// TIA Portal project "11_Sorting_Station" (V19)

(* hardware
DEVICE "S7-1500/ET200MP station_1"  S7-1500 station
   slot 0: "Rail_0"  Rack  6ES7 590-1***0-0AA0
   slot 1: "PLC_1"  CPU 1513-1 PN  6ES7 513-1AL02-0AB0  V2.9
      slot 3: "CPU display_1"  6ES7591-1AA00-0AA0
      slot 32768: "PROFINET interface_1"  X1
         slot 32769: "Port_1"  X1 P1
         slot 32770: "Port_2"  X1 P2
      slot 34817: "Virtual CP interface port_1"  Virtual CP interface port  Virtual CP interface port
*)

// ===== PLC "PLC_1"  CPU 1513-1 PN =====

VAR_GLOBAL   // PLC tag table "Default tag table"
   "nw2" AT %M0.0 : Bool;
   "nw3 2nd memory (Pause)" AT %M0.2 : Bool;
   "nw3 1st memory (Unpause)" AT %M0.1 : Bool;
   "nw4" AT %M0.5 : Bool;
   "nw4 Vision sensor O/P" AT %M0.6 : Bool;
   "nw5" AT %M0.3 : Bool;
   "nw5 VS O/P N" AT %M0.7 : Bool;
   "nw6" AT %M0.4 : Bool;
   "nw7" AT %M1.0 : Bool;
   "nw10" AT %M1.3 : Bool;
   "nw10 s1t N" AT %M1.4 : Bool;
   "nw11" AT %M1.5 : Bool;
   "nw11 s2t N" AT %M1.6 : Bool;
   "nw12" AT %M1.7 : Bool;
   "nw12 s2t N" AT %M2.0 : Bool;
   "nw8" AT %M1.1 : Bool;
   "nw9" AT %M1.2 : Bool;
END_VAR

VAR_GLOBAL   // PLC tag table "Tag table from XML_1"
   "Start" AT %I0.0 : Bool;
   "Pause & Unpause" AT %I0.1 : Bool;
   "Reset" AT %I0.2 : Bool;
   "At exit" AT %I0.3 : Bool;
   "Start light" AT %Q0.0 : Bool;
   "Pause & U Light" AT %Q0.1 : Bool;
   "Reset light" AT %Q0.2 : Bool;
   "Entry conveyor" AT %Q0.3 : Bool;
   "Exit conveyor" AT %Q0.4 : Bool;
   "Sorter 1 belt" AT %Q0.5 : Bool;
   "Sorter 1 turn" AT %Q0.6 : Bool;
   "Sorter 2 belt" AT %Q0.7 : Bool;
   "Sorter 2 turn" AT %Q1.0 : Bool;
   "Sorter 3 belt" AT %Q1.1 : Bool;
   "Sorter 3 turn" AT %Q1.2 : Bool;
   "Vision sensor" AT %ID30 : DInt;
   "Raw Materials Count" AT %QD30 : DInt;
   "Product Base Count" AT %QD34 : DInt;
   "Product Lid Count" AT %QD38 : DInt;
END_VAR

// folder: System blocks/Program resources

DATA_BLOCK "IEC_Counter_0_DB"   // DB1
{ S7_Optimized_Access := 'TRUE' }
AUTHOR : Simatic
FAMILY : IEC
NAME : CNTR
VERSION : 1.0
// stored: InstanceOfName IEC_COUNTER
"IEC_COUNTER"
BEGIN
END_DATA_BLOCK

DATA_BLOCK "IEC_Counter_0_DB_1"   // DB2
{ S7_Optimized_Access := 'TRUE' }
AUTHOR : Simatic
FAMILY : IEC
NAME : CNTR
VERSION : 1.0
// stored: InstanceOfName IEC_COUNTER
"IEC_COUNTER"
BEGIN
END_DATA_BLOCK

DATA_BLOCK "IEC_Counter_0_DB_2"   // DB3
{ S7_Optimized_Access := 'TRUE' }
AUTHOR : Simatic
FAMILY : IEC
NAME : CNTR
VERSION : 1.0
// stored: InstanceOfName IEC_COUNTER
"IEC_COUNTER"
BEGIN
END_DATA_BLOCK

// folder: (top level)

ORGANIZATION_BLOCK "Main"   // OB1, LAD, ProgramCycle
TITLE = "Main Program Sweep (Cycle)"
{ S7_Optimized_Access := 'TRUE' }
VERSION : 0.1
   VAR_INPUT
      Initial_Call : Bool;   // Initial call of this OB
      Remanence : Bool;   // =True, if remanent data are available
   END_VAR
   VAR_TEMP   // added for the SCL form of the ladder/FBD networks
      _w1 : Bool;
   END_VAR
BEGIN

REGION Network 2: Start/Reset system
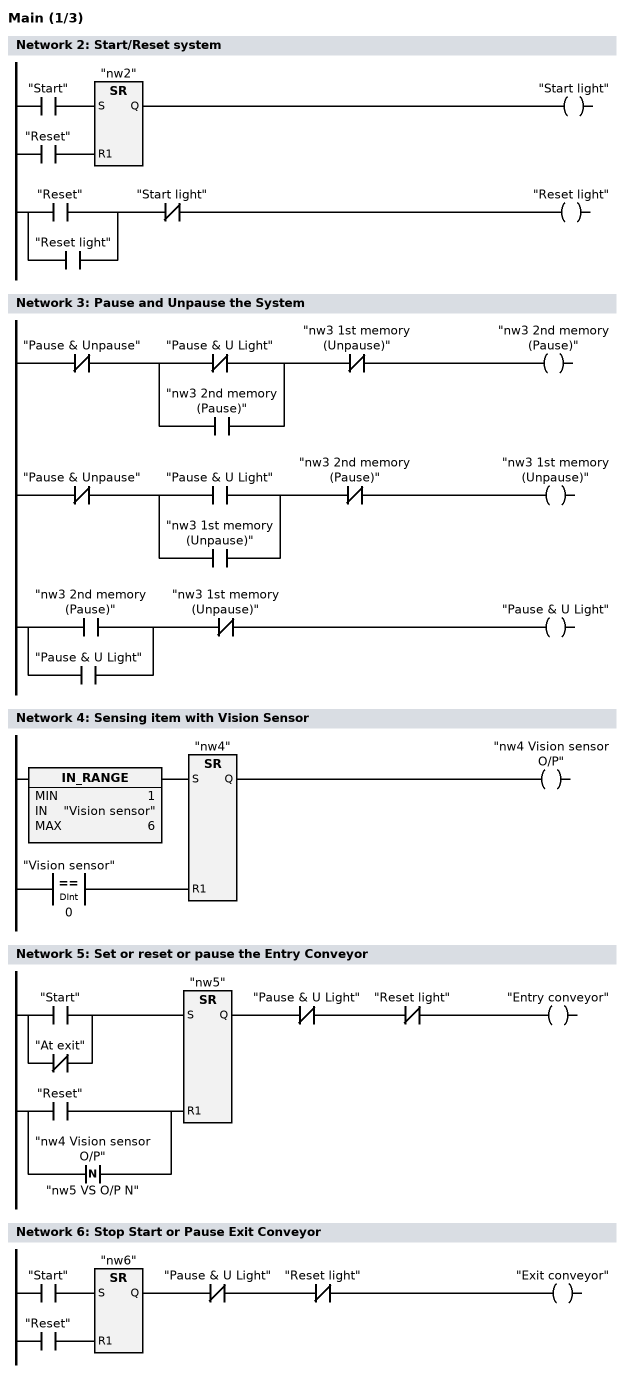
   RUNG wire#powerrail
      Contact( "Start" )
      S_SR(operand := "nw2", r1 := wire#w1)
      Coil( "Start light" )
   END_RUNG
   RUNG wire#powerrail
      Contact( "Reset" )
   END_RUNG wire#w1
   RUNG wire#powerrail
      Contact( "Reset" )
      wire#w2
      I_Contact( "Start light" )
      Coil( "Reset light" )
   END_RUNG
   RUNG wire#powerrail
      Contact( "Reset light" )
   END_RUNG wire#w2
   // the same network as SCL:
   IF "Start" THEN
       "nw2" := TRUE;   // SR flip-flop
   END_IF;
   IF "Reset" THEN "nw2" := FALSE; END_IF;
   "Start light" := "nw2";
   "Reset light" := ("Reset" OR "Reset light") AND NOT "Start light";
END_REGION

REGION Network 3: Pause and Unpause the System
   RUNG wire#powerrail
      I_Contact( "Pause & Unpause" )
      wire#w1
      I_Contact( "Pause & U Light" )
      wire#w2
      I_Contact( "nw3 1st memory (Unpause)" )
      Coil( "nw3 2nd memory (Pause)" )
   END_RUNG
   RUNG wire#w1
      Contact( "nw3 2nd memory (Pause)" )
   END_RUNG wire#w2
   RUNG wire#powerrail
      I_Contact( "Pause & Unpause" )
      wire#w3
      Contact( "Pause & U Light" )
      wire#w4
      I_Contact( "nw3 2nd memory (Pause)" )
      Coil( "nw3 1st memory (Unpause)" )
   END_RUNG
   RUNG wire#w3
      Contact( "nw3 1st memory (Unpause)" )
   END_RUNG wire#w4
   RUNG wire#powerrail
      Contact( "nw3 2nd memory (Pause)" )
      wire#w5
      I_Contact( "nw3 1st memory (Unpause)" )
      Coil( "Pause & U Light" )
   END_RUNG
   RUNG wire#powerrail
      Contact( "Pause & U Light" )
   END_RUNG wire#w5
   // the same network as SCL:
   "nw3 2nd memory (Pause)" := NOT "Pause & Unpause" AND (NOT "Pause & U Light" OR "nw3 2nd memory (Pause)") AND NOT "nw3 1st memory (Unpause)";
   "nw3 1st memory (Unpause)" := NOT "Pause & Unpause" AND ("Pause & U Light" OR "nw3 1st memory (Unpause)") AND NOT "nw3 2nd memory (Pause)";
   "Pause & U Light" := ("nw3 2nd memory (Pause)" OR "Pause & U Light") AND NOT "nw3 1st memory (Unpause)";
END_REGION

REGION Network 4: Sensing item with Vision Sensor
   RUNG wire#powerrail
      { S7_Templates := "SrcType := DInt" } InRange(min := 1, in := "Vision sensor", max := 6)
      S_SR(operand := "nw4", r1 := wire#w1)
      Coil( "nw4 Vision sensor O/P" )
   END_RUNG
   RUNG wire#powerrail
      { S7_Templates := "SrcType := DInt" } EQ_Contact(in1 := "Vision sensor", in2 := 0)
   END_RUNG wire#w1
   // the same network as SCL:
   IF (1 <= "Vision sensor") AND ("Vision sensor" <= 6) THEN
       "nw4" := TRUE;   // SR flip-flop
   END_IF;
   IF "Vision sensor" = 0 THEN "nw4" := FALSE; END_IF;
   "nw4 Vision sensor O/P" := "nw4";
END_REGION

REGION Network 5: Set or reset or pause the Entry Conveyor
   RUNG wire#powerrail
      Contact( "Start" )
      wire#w1
      S_SR(operand := "nw5", r1 := wire#w2)
      I_Contact( "Pause & U Light" )
      I_Contact( "Reset light" )
      Coil( "Entry conveyor" )
   END_RUNG
   RUNG wire#powerrail
      I_Contact( "At exit" )
   END_RUNG wire#w1
   RUNG wire#powerrail
      Contact( "Reset" )
   END_RUNG wire#w2
   RUNG wire#powerrail
      N_Contact(operand := "nw4 Vision sensor O/P", bit := "nw5 VS O/P N")
   END_RUNG wire#w2
   // the same network as SCL:
   #_w1 := NOT "nw4 Vision sensor O/P" AND "nw5 VS O/P N";   // falling edge of "nw4 Vision sensor O/P"
   "nw5 VS O/P N" := "nw4 Vision sensor O/P";
   IF "Start" OR NOT "At exit" THEN
       "nw5" := TRUE;   // SR flip-flop
   END_IF;
   IF "Reset" OR #_w1 THEN "nw5" := FALSE; END_IF;
   "Entry conveyor" := "nw5" AND NOT "Pause & U Light" AND NOT "Reset light";
END_REGION

REGION Network 6: Stop Start or Pause Exit Conveyor
   RUNG wire#powerrail
      Contact( "Start" )
      S_SR(operand := "nw6", r1 := wire#w1)
      I_Contact( "Pause & U Light" )
      I_Contact( "Reset light" )
      Coil( "Exit conveyor" )
   END_RUNG
   RUNG wire#powerrail
      Contact( "Reset" )
   END_RUNG wire#w1
   // the same network as SCL:
   IF "Start" THEN
       "nw6" := TRUE;   // SR flip-flop
   END_IF;
   IF "Reset" THEN "nw6" := FALSE; END_IF;
   "Exit conveyor" := "nw6" AND NOT "Pause & U Light" AND NOT "Reset light";
END_REGION

REGION Network 7: Set/Reset/Pause for Sorter 1, which is RAW_MATERIALS
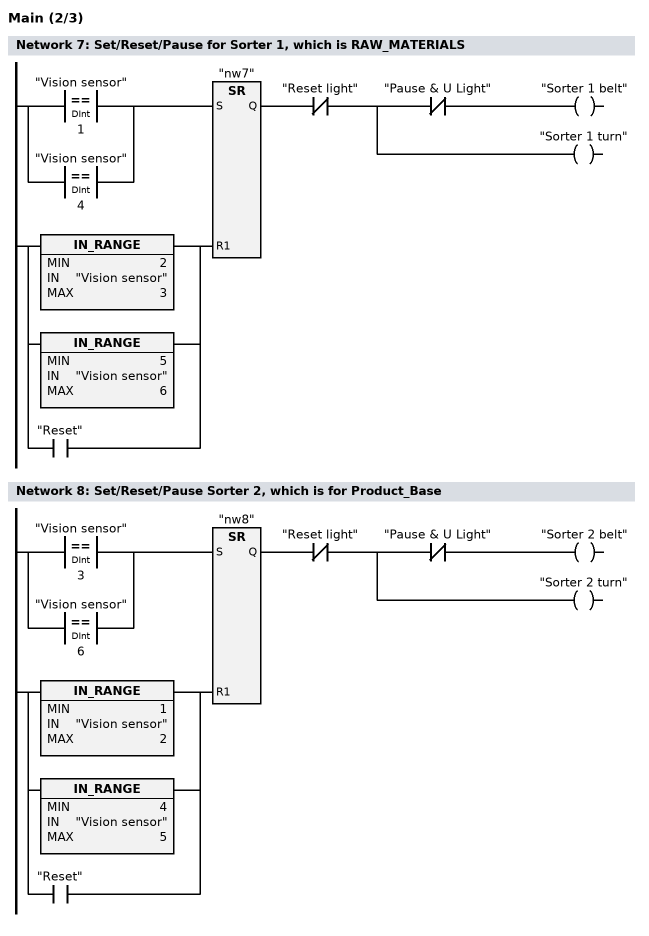
   RUNG wire#powerrail
      { S7_Templates := "SrcType := DInt" } EQ_Contact(in1 := "Vision sensor", in2 := 1)
      wire#w1
      S_SR(operand := "nw7", r1 := wire#w2)
      I_Contact( "Reset light" )
      wire#w3
      I_Contact( "Pause & U Light" )
      Coil( "Sorter 1 belt" )
   END_RUNG
   RUNG wire#powerrail
      { S7_Templates := "SrcType := DInt" } EQ_Contact(in1 := "Vision sensor", in2 := 4)
   END_RUNG wire#w1
   RUNG wire#powerrail
      { S7_Templates := "SrcType := DInt" } InRange(min := 2, in := "Vision sensor", max := 3)
   END_RUNG wire#w2
   RUNG wire#powerrail
      { S7_Templates := "SrcType := DInt" } InRange(min := 5, in := "Vision sensor", max := 6)
   END_RUNG wire#w2
   RUNG wire#powerrail
      Contact( "Reset" )
   END_RUNG wire#w2
   RUNG wire#w3
      Coil( "Sorter 1 turn" )
   END_RUNG
   // the same network as SCL:
   IF ("Vision sensor" = 1) OR ("Vision sensor" = 4) THEN
       "nw7" := TRUE;   // SR flip-flop
   END_IF;
   IF ((2 <= "Vision sensor") AND ("Vision sensor" <= 3)) OR ((5 <= "Vision sensor") AND ("Vision sensor" <= 6)) OR "Reset" THEN
       "nw7" := FALSE;
   END_IF;
   #_w1 := "nw7" AND NOT "Reset light";
   "Sorter 1 belt" := #_w1 AND NOT "Pause & U Light";
   "Sorter 1 turn" := #_w1;
END_REGION

REGION Network 8: Set/Reset/Pause Sorter 2, which is for Product_Base
   RUNG wire#powerrail
      { S7_Templates := "SrcType := DInt" } EQ_Contact(in1 := "Vision sensor", in2 := 3)
      wire#w1
      S_SR(operand := "nw8", r1 := wire#w2)
      I_Contact( "Reset light" )
      wire#w3
      I_Contact( "Pause & U Light" )
      Coil( "Sorter 2 belt" )
   END_RUNG
   RUNG wire#powerrail
      { S7_Templates := "SrcType := DInt" } EQ_Contact(in1 := "Vision sensor", in2 := 6)
   END_RUNG wire#w1
   RUNG wire#powerrail
      { S7_Templates := "SrcType := DInt" } InRange(min := 1, in := "Vision sensor", max := 2)
   END_RUNG wire#w2
   RUNG wire#powerrail
      { S7_Templates := "SrcType := DInt" } InRange(min := 4, in := "Vision sensor", max := 5)
   END_RUNG wire#w2
   RUNG wire#powerrail
      Contact( "Reset" )
   END_RUNG wire#w2
   RUNG wire#w3
      Coil( "Sorter 2 turn" )
   END_RUNG
   // the same network as SCL:
   IF ("Vision sensor" = 3) OR ("Vision sensor" = 6) THEN
       "nw8" := TRUE;   // SR flip-flop
   END_IF;
   IF ((1 <= "Vision sensor") AND ("Vision sensor" <= 2)) OR ((4 <= "Vision sensor") AND ("Vision sensor" <= 5)) OR "Reset" THEN
       "nw8" := FALSE;
   END_IF;
   #_w1 := "nw8" AND NOT "Reset light";
   "Sorter 2 belt" := #_w1 AND NOT "Pause & U Light";
   "Sorter 2 turn" := #_w1;
END_REGION

REGION Network 9: Set/Reset/Pause Sorter 3, which is for Product_Lid
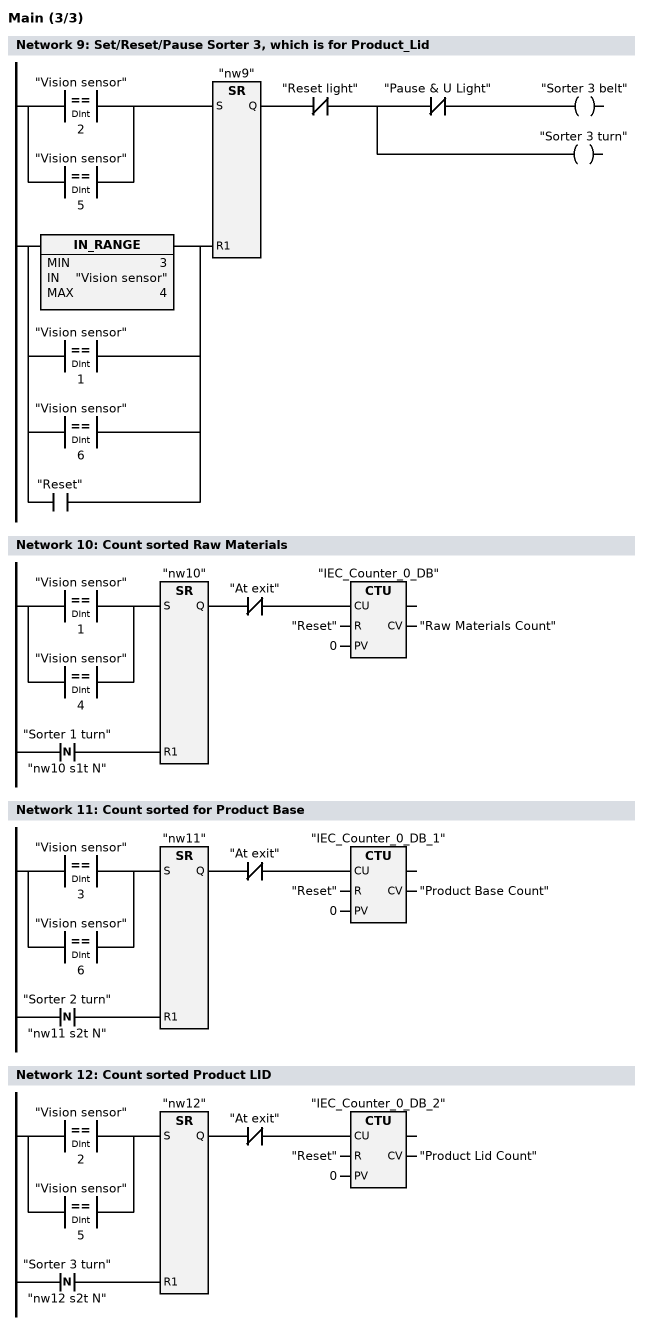
   RUNG wire#powerrail
      { S7_Templates := "SrcType := DInt" } EQ_Contact(in1 := "Vision sensor", in2 := 2)
      wire#w1
      S_SR(operand := "nw9", r1 := wire#w2)
      I_Contact( "Reset light" )
      wire#w3
      I_Contact( "Pause & U Light" )
      Coil( "Sorter 3 belt" )
   END_RUNG
   RUNG wire#powerrail
      { S7_Templates := "SrcType := DInt" } EQ_Contact(in1 := "Vision sensor", in2 := 5)
   END_RUNG wire#w1
   RUNG wire#powerrail
      { S7_Templates := "SrcType := DInt" } InRange(min := 3, in := "Vision sensor", max := 4)
   END_RUNG wire#w2
   RUNG wire#powerrail
      { S7_Templates := "SrcType := DInt" } EQ_Contact(in1 := "Vision sensor", in2 := 1)
   END_RUNG wire#w2
   RUNG wire#powerrail
      { S7_Templates := "SrcType := DInt" } EQ_Contact(in1 := "Vision sensor", in2 := 6)
   END_RUNG wire#w2
   RUNG wire#powerrail
      Contact( "Reset" )
   END_RUNG wire#w2
   RUNG wire#w3
      Coil( "Sorter 3 turn" )
   END_RUNG
   // the same network as SCL:
   IF ("Vision sensor" = 2) OR ("Vision sensor" = 5) THEN
       "nw9" := TRUE;   // SR flip-flop
   END_IF;
   IF ((3 <= "Vision sensor") AND ("Vision sensor" <= 4)) OR ("Vision sensor" = 1) OR ("Vision sensor" = 6) OR "Reset" THEN
       "nw9" := FALSE;
   END_IF;
   #_w1 := "nw9" AND NOT "Reset light";
   "Sorter 3 belt" := #_w1 AND NOT "Pause & U Light";
   "Sorter 3 turn" := #_w1;
END_REGION

REGION Network 10: Count sorted Raw Materials
   #_w1 := NOT "Sorter 1 turn" AND "nw10 s1t N";   // falling edge of "Sorter 1 turn"
   "nw10 s1t N" := "Sorter 1 turn";
   IF ("Vision sensor" = 1) OR ("Vision sensor" = 4) THEN
       "nw10" := TRUE;   // SR flip-flop
   END_IF;
   IF #_w1 THEN "nw10" := FALSE; END_IF;
   "IEC_Counter_0_DB".CTU(CU := "nw10" AND NOT "At exit", R := "Reset", PV := 0, CV => "Raw Materials Count");
END_REGION

REGION Network 11: Count sorted for Product Base
   #_w1 := NOT "Sorter 2 turn" AND "nw11 s2t N";   // falling edge of "Sorter 2 turn"
   "nw11 s2t N" := "Sorter 2 turn";
   IF ("Vision sensor" = 3) OR ("Vision sensor" = 6) THEN
       "nw11" := TRUE;   // SR flip-flop
   END_IF;
   IF #_w1 THEN "nw11" := FALSE; END_IF;
   "IEC_Counter_0_DB_1".CTU(CU := "nw11" AND NOT "At exit", R := "Reset", PV := 0, CV => "Product Base Count");
END_REGION

REGION Network 12: Count sorted Product LID
   #_w1 := NOT "Sorter 3 turn" AND "nw12 s2t N";   // falling edge of "Sorter 3 turn"
   "nw12 s2t N" := "Sorter 3 turn";
   IF ("Vision sensor" = 2) OR ("Vision sensor" = 5) THEN
       "nw12" := TRUE;   // SR flip-flop
   END_IF;
   IF #_w1 THEN "nw12" := FALSE; END_IF;
   "IEC_Counter_0_DB_2".CTU(CU := "nw12" AND NOT "At exit", R := "Reset", PV := 0, CV => "Product Lid Count");
END_REGION
END_ORGANIZATION_BLOCK